FUNCTION_BLOCK Manipulator (* Basic Function Block Type *)
  (* Standard: 61499-2 *)
  (* Version 0.0, 2015-03-26, 4DIAC-IDE, 4DIAC-Consortium *)
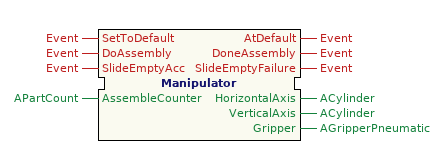
  EVENT_INPUT
    SetToDefault;
    DoAssembly;
    SlideEmptyAcc;
  END_EVENT
  EVENT_OUTPUT
    AtDefault;
    DoneAssembly;
    SlideEmptyFailure;
  END_EVENT
  SOCKETS
    AssembleCounter : APartCount;
  END_SOCKETS
  PLUGS
    HorizontalAxis : ACylinder;
    VerticalAxis : ACylinder;
    Gripper : AGripperPneumatic;
  END_PLUGS
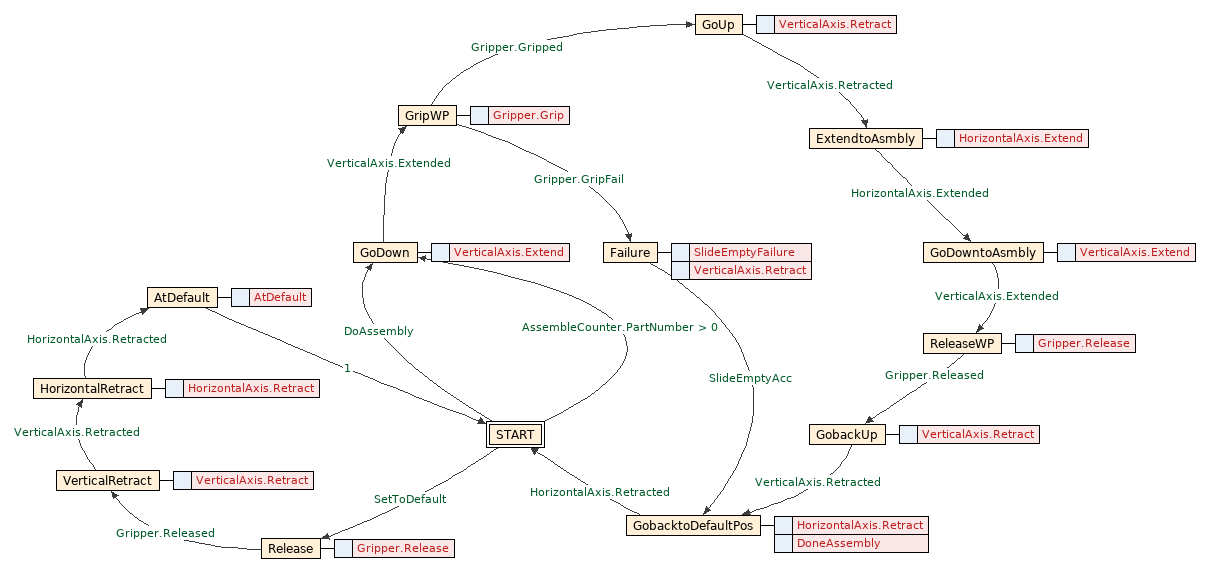
  EC_STATES
    START; (* Initial State *)
    Release : -> Gripper.Release; (* Initialization *)
    VerticalRetract : -> VerticalAxis.Retract;
    HorizontalRetract : -> HorizontalAxis.Retract;
    GoDown : -> VerticalAxis.Extend;
    GripWP : -> Gripper.Grip;
    GoUp : -> VerticalAxis.Retract;
    ExtendtoAsmbly : -> HorizontalAxis.Extend;
    GoDowntoAsmbly : -> VerticalAxis.Extend;
    ReleaseWP : -> Gripper.Release;
    GobackUp : -> VerticalAxis.Retract;
    GobacktoDefaultPos : -> HorizontalAxis.Retract, -> DoneAssembly;
    Failure : -> SlideEmptyFailure, -> VerticalAxis.Retract;
    AtDefault : -> AtDefault;
  END_STATES
  EC_TRANSITIONS
    START TO Release := SetToDefault;
    Release TO VerticalRetract := Gripper.Released;
    VerticalRetract TO HorizontalRetract := VerticalAxis.Retracted;
    START TO GoDown := DoAssembly;
    GoDown TO GripWP := VerticalAxis.Extended;
    GripWP TO GoUp := Gripper.Gripped;
    GoUp TO ExtendtoAsmbly := VerticalAxis.Retracted;
    GoDowntoAsmbly TO ReleaseWP := VerticalAxis.Extended;
    ReleaseWP TO GobackUp := Gripper.Released;
    GobackUp TO GobacktoDefaultPos := VerticalAxis.Retracted;
    ExtendtoAsmbly TO GoDowntoAsmbly := HorizontalAxis.Extended;
    GripWP TO Failure := Gripper.GripFail;
    GobacktoDefaultPos TO START := HorizontalAxis.Retracted;
    HorizontalRetract TO AtDefault := HorizontalAxis.Retracted;
    AtDefault TO START := 1;
    START TO GoDown := AssembleCounter.PartNumber > 0;
    Failure TO GobacktoDefaultPos := SlideEmptyAcc;
  END_TRANSITIONS
END_FUNCTION_BLOCK
